TYPE ST_GearInPos : //
STRUCT
	bEnable		                        :BOOL;	
   	bEnable2                       :BOOL;	

	bGearOutMode                 :BOOL;
    fMasterSyncPosition           :LREAL;  
    fSlaveSyncPosition              :LREAL;  

	bReady                            :BOOL;  
    bStartSync		 	               :BOOL;	
	bInSync		 	                   :BOOL;	
    bBusy                               :BOOL;	
	bError				               :BOOL;		

END_STRUCT
END_TYPE

(* stored: Version 1.1.0.1, ProductVersion 3.1.4024.9
   DUT ST_GearInPos: Id {35fd5f5f-8858-44fd-a45a-35aee093406f} *)
